TYPE ST_HMI_MANUAL_AXIS_ITEM :
STRUCT
	stName	: ST_Text;
	fPos	: REAL;
END_STRUCT
END_TYPE

(* stored: Version 1.1.0.1
   DUT ST_HMI_MANUAL_AXIS_ITEM: Id {44292beb-42c5-4fe1-9035-b97a86baf38d} *)
